// TIA Portal V15.1 export
// export: Created 2022-03-15T12:28:26.5433842Z, ExportSetting WithDefaults, WithReadOnly, DisplayName Totally Integrated Automation Portal, DisplayVersion V15.1 Update 3, DisplayName TIA Portal Openness, DisplayVersion V15.1, DisplayName TIA Portal Teamcenter Gateway, DisplayVersion V15.1, DisplayName SINAMICS Startdrive Advanced, DisplayVersion V15.1, DisplayName G130, G150, S120, S150, SINAMICS MV, S210, DisplayVersion V15.1, DisplayName G110M, G120, G120C, G120D, G120P, DisplayVersion V15.1, DisplayName STEP 7 Professional, DisplayVersion V15.1 Update 3, DisplayName STEP 7 Safety, DisplayVersion V15.1, DisplayName WinCC Advanced, DisplayVersion V15.1 Update 3
ORGANIZATION_BLOCK "Main"   // OB1, LAD, ProgramCycle
TITLE = "Main Program Sweep (Cycle)"
{ S7_Optimized_Access := 'TRUE' }
VERSION : 0.1
// stored: AutoNumber true, CodeModifiedDate 2022-03-08T11:13:54.5164113Z, CompileDate 2022-03-08T11:13:55.9851651Z, ConstantName OB_Main, CreationDate 2022-02-28T09:16:09.6965758Z, EventClass Program cycle, HandleErrorsWithinBlock false, InterfaceModifiedDate 2022-02-28T09:18:02.6969839Z, IsConsistent true, IsIECCheckEnabled false, IsKnowHowProtected false, IsWriteProtected false, ModifiedDate 2022-03-08T11:13:54.5164113Z, ParameterModified 2022-02-28T09:18:02.6969839Z, PLCSimAdvancedSupport false, PriorityNumber 1, ProcessImagePartNumber 65535, SetENOAutomatically False, StructureModified 2022-02-28T09:18:02.6969839Z
   VAR_INPUT
      Initial_Call : Bool;   // Initial call of this OB
      Remanence : Bool;   // =True, if remanent data are available
   END_VAR
BEGIN

REGION Network 1
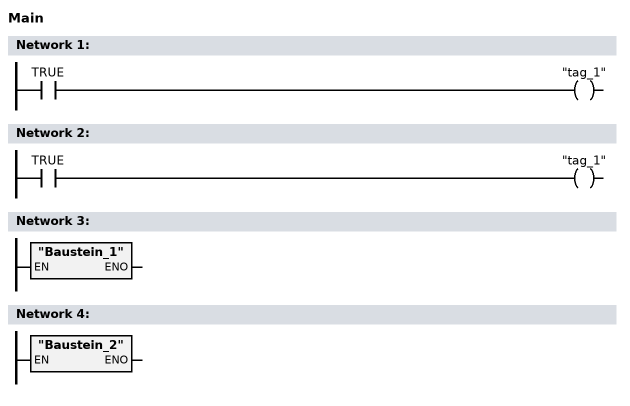
   RUNG wire#powerrail
      Contact( TRUE )
      Coil( "tag_1" )
   END_RUNG
   // the same network as SCL:
   "tag_1" := TRUE;
END_REGION

REGION Network 2
   RUNG wire#powerrail
      Contact( TRUE )
      Coil( "tag_1" )
   END_RUNG
   // the same network as SCL:
   "tag_1" := TRUE;
END_REGION

REGION Network 3
   RUNG wire#powerrail
      "Baustein_1"()
   END_RUNG
   // the same network as SCL:
   "Baustein_1"();
END_REGION

REGION Network 4
   RUNG wire#powerrail
      "Baustein_2"()
   END_RUNG
   // the same network as SCL:
   "Baustein_2"();
END_REGION
END_ORGANIZATION_BLOCK
